{attribute 'GeneratedUsingTerminal: ELX9560-0000-0016'}
{attribute addProperty BoxType "ELX9560-0000-0016"}
{attribute addProperty Id "Status_UinAT %I*Status_Uin_449D6AB51Status_UexAT %I*Status_Uex_449D6AB51WcStateAT %I*WcState_9091E0EB2InfoDataAT %I*InfoData_6F19DB2B2"}
{attribute addProperty CRC "2285638051"}
{attribute addProperty Size "6"}
TYPE ELX9560_883C11A3 EXTENDS EtcSlaveTerminalBase_947E5A46 :
STRUCT
	{attribute addProperty Name "Status_Uin"}
	Status_Uin : Status_Uin_449D6AB5;
	{attribute addProperty Name "Status_Uex"}
	Status_Uex : Status_Uex_449D6AB5;
	{attribute addProperty Name "WcState"}
	WcState : WcState_9091E0EB;
	{attribute addProperty Name "InfoData"}
	InfoData : InfoData_6F19DB2B;
END_STRUCT
END_TYPE

(* stored: Version 1.2.0.0, ProductVersion 3.1.4024.9
   DUT ELX9560_883C11A3: Id {9eddb27a-1515-4dfc-9c6e-49dbb54f24cc} *)
